  MoveL 5117 to (-316.66, 5.05, -299.32) mm, rotated rx -179.15 ry 0 rz -30.08 deg; joints [-2.67, -65.712, 120.564, -183.679, 54.716, 242.25]
  MoveC 5118 to (-316.6, 5.19, -299.32) mm, rotated rx -179.15 ry 0 rz -30.08 deg; joints [-2.667, -65.719, 120.562, -183.677, 54.707, 242.249] to (-316.58, 5.33, -299.32) mm, rotated rx -179.15 ry 0 rz -30.08 deg; joints [-2.666, -65.726, 120.559, -183.676, 54.697, 242.249]
  MoveL 5119 to (-316.58, 5.33, -299.32) mm, rotated rx -179.15 ry 0 rz -30.08 deg; joints [-2.666, -65.726, 120.559, -183.676, 54.697, 242.249]
  MoveC 5120 to (-316.55, 5.47, -299.32) mm, rotated rx -179.15 ry 0 rz -30.08 deg; joints [-2.665, -65.733, 120.557, -183.675, 54.688, 242.249] to (-316.49, 5.6, -299.32) mm, rotated rx -179.15 ry 0 rz -30.08 deg; joints [-2.662, -65.74, 120.555, -183.672, 54.679, 242.248]
  MoveL 5121 to (-316.49, 5.6, -299.32) mm, rotated rx -179.15 ry 0 rz -30.08 deg; joints [-2.662, -65.74, 120.555, -183.672, 54.679, 242.248]
  MoveC 5122 to (-315.82, 6.77, -299.88) mm, rotated rx -179.15 ry 0 rz -30.08 deg; joints [-2.632, -65.771, 120.491, -183.638, 54.584, 242.233] to (-315.54, 7.25, -301.23) mm, rotated rx -179.15 ry 0 rz -30.08 deg; joints [-2.617, -65.725, 120.375, -183.623, 54.512, 242.228]
  MoveL 5123 to (-315.54, 7.25, -301.23) mm, rotated rx -179.15 ry 0 rz -30.08 deg; joints [-2.617, -65.725, 120.375, -183.623, 54.512, 242.228]
  MoveL 5124 to (-315.54, 7.25, -303.77) mm, rotated rx -179.15 ry 0 rz -30.08 deg; joints [-2.612, -65.594, 120.169, -183.62, 54.438, 242.23]
  MoveC 5125 to (-315.82, 6.77, -305.11) mm, rotated rx -179.15 ry 0 rz -30.08 deg; joints [-2.621, -65.499, 120.067, -183.633, 54.431, 242.238] to (-316.49, 5.6, -305.67) mm, rotated rx -179.15 ry 0 rz -30.08 deg; joints [-2.65, -65.411, 120.04, -183.665, 54.493, 242.253]
  MoveL 5126 to (-316.49, 5.6, -305.67) mm, rotated rx -179.15 ry 0 rz -30.08 deg; joints [-2.65, -65.411, 120.04, -183.665, 54.493, 242.253]
  MoveC 5127 to (-316.55, 5.47, -305.67) mm, rotated rx -179.15 ry 0 rz -30.08 deg; joints [-2.652, -65.404, 120.042, -183.668, 54.502, 242.254] to (-316.58, 5.33, -305.67) mm, rotated rx -179.15 ry 0 rz -30.08 deg; joints [-2.654, -65.397, 120.045, -183.669, 54.512, 242.255]
  MoveL 5128 to (-316.58, 5.33, -305.67) mm, rotated rx -179.15 ry 0 rz -30.08 deg; joints [-2.654, -65.397, 120.045, -183.669, 54.512, 242.255]
  MoveC 5129 to (-316.6, 5.18, -305.67) mm, rotated rx -179.15 ry 0 rz -30.08 deg; joints [-2.655, -65.39, 120.047, -183.67, 54.521, 242.255] to (-316.66, 5.05, -305.67) mm, rotated rx -179.15 ry 0 rz -30.08 deg; joints [-2.657, -65.383, 120.049, -183.672, 54.53, 242.256]
  MoveL 5130 to (-316.66, 5.05, -305.67) mm, rotated rx -179.15 ry 0 rz -30.08 deg; joints [-2.657, -65.383, 120.049, -183.672, 54.53, 242.256]
  MoveL 5131 to (-327.16, -13.08, -305.67) mm, rotated rx -179.15 ry 0 rz -30.08 deg; joints [-3.118, -64.446, 120.311, -184.177, 55.745, 242.475]
  MoveC 5132 to (-327.25, -13.19, -305.67) mm, rotated rx -179.15 ry 0 rz -30.08 deg; joints [-3.122, -64.44, 120.313, -184.181, 55.752, 242.477] to (-327.36, -13.29, -305.67) mm, rotated rx -179.15 ry 0 rz -30.08 deg; joints [-3.127, -64.435, 120.314, -184.186, 55.759, 242.48]
  MoveL 5133 to (-327.36, -13.29, -305.67) mm, rotated rx -179.15 ry 0 rz -30.08 deg; joints [-3.127, -64.435, 120.314, -184.186, 55.759, 242.48]
  MoveC 5134 to (-327.47, -13.38, -305.67) mm, rotated rx -179.15 ry 0 rz -30.08 deg; joints [-3.132, -64.43, 120.315, -184.192, 55.765, 242.483] to (-327.55, -13.5, -305.67) mm, rotated rx -179.15 ry 0 rz -30.08 deg; joints [-3.136, -64.424, 120.316, -184.196, 55.773, 242.484]
  MoveL 5135 to (-327.55, -13.5, -305.67) mm, rotated rx -179.15 ry 0 rz -30.08 deg; joints [-3.136, -64.424, 120.316, -184.196, 55.773, 242.484]
  MoveC 5136 to (-328.23, -14.66, -306.23) mm, rotated rx -179.15 ry 0 rz -30.08 deg; joints [-3.164, -64.334, 120.287, -184.227, 55.833, 242.498] to (-328.51, -15.14, -307.58) mm, rotated rx -179.15 ry 0 rz -30.08 deg; joints [-3.173, -64.241, 120.183, -184.239, 55.824, 242.505]
  MoveL 5137 to (-328.51, -15.14, -307.58) mm, rotated rx -179.15 ry 0 rz -30.08 deg; joints [-3.173, -64.241, 120.183, -184.239, 55.824, 242.505]
  MoveL 5138 to (-328.51, -15.14, -310.11) mm, rotated rx -179.15 ry 0 rz -30.08 deg; joints [-3.167, -64.112, 119.976, -184.236, 55.746, 242.508]
  MoveC 5139 to (-328.23, -14.66, -311.46) mm, rotated rx -179.15 ry 0 rz -30.08 deg; joints [-3.152, -64.069, 119.86, -184.221, 55.672, 242.504] to (-327.55, -13.5, -312.02) mm, rotated rx -179.15 ry 0 rz -30.08 deg; joints [-3.121, -64.101, 119.799, -184.188, 55.578, 242.492]
  MoveL 5140 to (-327.55, -13.5, -312.02) mm, rotated rx -179.15 ry 0 rz -30.08 deg; joints [-3.121, -64.101, 119.799, -184.188, 55.578, 242.492]
  MoveL 5141 to (-327.53, -13.46, -312.02) mm, rotated rx -179.15 ry 0 rz -30.08 deg; joints [-3.12, -64.103, 119.799, -184.187, 55.575, 242.491]
  MoveC 5142 to (-327.45, -13.34, -312.02) mm, rotated rx -179.15 ry 0 rz -30.08 deg; joints [-3.116, -64.109, 119.797, -184.183, 55.567, 242.489] to (-327.34, -13.25, -312.02) mm, rotated rx -179.15 ry 0 rz -30.08 deg; joints [-3.111, -64.115, 119.796, -184.177, 55.561, 242.486]
  MoveL 5143 to (-327.34, -13.25, -312.02) mm, rotated rx -179.15 ry 0 rz -30.08 deg; joints [-3.111, -64.115, 119.796, -184.177, 55.561, 242.486]
  MoveC 5144 to (-327.23, -13.15, -312.02) mm, rotated rx -179.15 ry 0 rz -30.08 deg; joints [-3.106, -64.12, 119.795, -184.172, 55.555, 242.484] to (-327.14, -13.04, -312.02) mm, rotated rx -179.15 ry 0 rz -30.08 deg; joints [-3.103, -64.126, 119.794, -184.167, 55.547, 242.482]
  MoveL 5145 to (-327.14, -13.04, -312.02) mm, rotated rx -179.15 ry 0 rz -30.08 deg; joints [-3.103, -64.126, 119.794, -184.167, 55.547, 242.482]
  MoveL 5146 to (-316.99, 4.48, -312.02) mm, rotated rx -179.15 ry 0 rz -30.08 deg; joints [-2.659, -65.025, 119.542, -183.682, 54.381, 242.269]
  MoveC 5147 to (-316.87, 5.44, -312.02) mm, rotated rx -179.15 ry 0 rz -30.08 deg; joints [-2.654, -65.073, 119.525, -183.678, 54.317, 242.27] to (-317.46, 6.21, -312.02) mm, rotated rx -179.15 ry 0 rz -30.08 deg; joints [-2.68, -65.109, 119.51, -183.712, 54.266, 242.293]
  MoveL 5148 to (-317.46, 6.21, -312.02) mm, rotated rx -179.15 ry 0 rz -30.08 deg; joints [-2.68, -65.109, 119.51, -183.712, 54.266, 242.293]
  Set speed (1000.0 mm/s)
  MoveL 5149 to (-338.78, 18.57, -312.02) mm, rotated rx -179.15 ry 0 rz -30.08 deg; joints [-3.617, -65.649, 119.195, -184.919, 53.456, 243.053]
  MoveL 5150 to (-338.78, 18.57, -312.02) mm, rotated rx -179.15 ry 0 rz -30.08 deg; joints [-3.617, -65.649, 119.195, -184.919, 53.456, 243.053]
